FUNCTION_BLOCK RunBridge EXTENDS RunUnitSlave
VAR_INPUT
	fakeAck AT%M* : BOOL;
END_VAR
VAR_OUTPUT
END_VAR
VAR
	bridge : defHandshake;
END_VAR

//----------------------------------------------
//	Bridge working signal and handshaking signal
//----------------------------------------------
SUPER^();

CASE outputState OF 
	//--------------------------------
	//	Initialization
	//--------------------------------	
	eSpecialStates.INITIAL_BEGIN:
		bridge.ready := FALSE;
		fakeAck:=FALSE;
		bSerialTransition := NOT bridge.ack AND NOT bridge.valid;
		IF bSerialTransition THEN
			NextState := eSpecialStates.INITIAL_END;
		END_IF
	//---------------------------------
	//	Working
	//---------------------------------
	eSpecialStates.SLAVE_ENTER_PROCEDURE:
		bridge.ready := TRUE;
		bSerialTransition := TRUE;
	16#201:
		bSerialTransition := bridge.ack OR fakeAck;
		IF bSerialTransition THEN
			fakeAck := FALSE; //auto-reset
			bridge.ready := FALSE;
		END_IF
	16#202:
		IF NOT bridge.ack THEN
			NextState := eSpecialStates.SLAVE_WORK_DONE;
		END_IF
END_CASE

END_FUNCTION_BLOCK

(* stored: Version 1.1.0.1, ProductVersion 3.1.4024.0
   POU RunBridge: Id {8efd5c53-7e74-4af7-97a5-3ec0eb5ea0d4}, SpecialFunc None *)
